TYPE ST_MachineParam :
STRUCT
	
END_STRUCT
END_TYPE

(* stored: Version 1.1.0.1, ProductVersion 3.1.4020.12
   DUT ST_MachineParam: Id {c80b1f56-f13d-4209-88a4-0f23a89dd9e9} *)
